Staubli VAL3: PCData.pjx

--- PCData.pjx ---
Parameters version=s7.3.1 stackSize=5000 millimeterUnit=true
Program file=start.pgx
Program file=stop.pgx
Data file=PCData.dtx

--- PCData.dtx ---
mdesc mNomSpeed
public frame fFrame = {fatherId=world[0]}
public num nNum[2]
public pointRx pPos[2]
  [0] = {fatherId=world[0]}
  [1] = {fatherId=world[0]}
public string sString
public trsf trTrsf[2]
public tool tTool[2]
  [0] = {fatherId=flange[0], ioLink=valve1}
  [1] = {fatherId=flange[0], ioLink=valve1}
public jointRx jJ[2]
public bool bBool

--- start.pgx ---
program start()
begin
  //*******************************************
  //Name: TestSoap
  //Function: test soap function
  //2012.05.28
  //y.ye@staubli.com
  //说明：这个作为一个库，被TestSoap调用
  //通过全局变量来与上位机进行交互
  //全局变量必须设定为public
  //*******************************************
end
